Staubli VAL3: restartMotor.pgx

program restartMotor()
begin
  restartMove()
  message="restartMove:done"
  taskCreate "sendStatus",100,sendStatus()
  taskKill ("restartMotor")
end
